FUNCTION_BLOCK ConveyorCTLRing (* Basic Function Block Type *)
  (* Standard: 61499-2 *)
  (* Version 0.2, 2003-12-04, JHC, Rockwell Automation, Renamed for better indexing. *)
  (* Version 0.1, 2002-11-05, JHC, Rockwell Automation, Corrected missing ST element in Algorithm REQ. *)
  (* Version 0.0, 2000-05-30, JHC, Rockwell Automation *)
  (* Compiler header: package fb.rt.cs725; *)
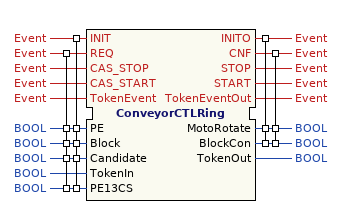
  EVENT_INPUT
    INIT WITH PE, Block, Candidate, PE13CS; (* Initialization Request *)
    REQ WITH PE, Block, Candidate, PE13CS; (* Normal Execution Request *)
    CAS_STOP;
    CAS_START;
    TokenEvent;
  END_EVENT
  EVENT_OUTPUT
    INITO WITH MotoRotate, BlockCon; (* Initialization Confirm *)
    CNF WITH MotoRotate, BlockCon; (* Execution Confirmation *)
    STOP;
    START;
    TokenEventOut;
  END_EVENT
  VAR_INPUT
    PE : BOOL; (* Input event qualifier *)
    Block : BOOL;
    Candidate : BOOL;
    TokenIn : BOOL;
    PE13CS : BOOL;
  END_VAR
  VAR_OUTPUT
    MotoRotate : BOOL; (* Output event qualifier *)
    BlockCon : BOOL;
    TokenOut : BOOL;
  END_VAR
  VAR
    lastPE : BOOL := 1;
    lastBlock : BOOL := 0;
  END_VAR
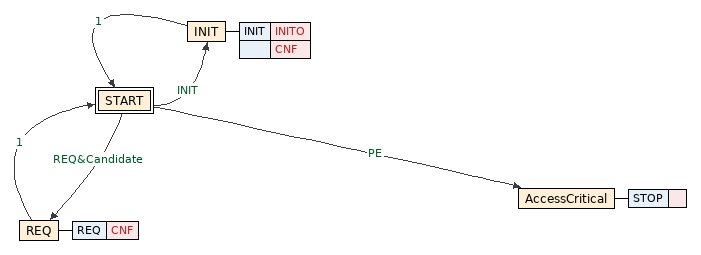
  EC_STATES
    START; (* Initial State *)
    INIT : INIT -> INITO, -> CNF; (* Initialization *)
    REQ : REQ -> CNF; (* Normal execution *)
    AccessCritical : STOP;
  END_STATES
  EC_TRANSITIONS
    START TO INIT := INIT;
    INIT TO START := 1;
    START TO REQ := REQ&Candidate;
    REQ TO START := 1;
    START TO AccessCritical := PE;
  END_TRANSITIONS
  ALGORITHM INIT IN ST: (* Initialization algorithm *)
MotoRotate := TRUE;
Block := FALSE;

System.out.println(this + " " + MotoRotate);
System.out.println(MotoRotate);
  END_ALGORITHM
  ALGORITHM REQ IN Java: (* Normally executed algorithm *)
System.out.println(this+" -> Candidate"+Candidate.value);
if(Candidate.value){
if(lastPE.value!=PE.value){
if(!PE.value){
BlockCon.value=true;
System.out.println("BlockCon = true");
}
else{
BlockCon.value=false;
System.out.println("BlockCon = false");
}
lastPE.value=PE.value;
}
if(lastBlock.value!=Block.value){
if(Block.value){
STOP.serviceEvent(this);
MotoRotate.value=false;
System.out.println("Cas Stop");
}
else{
START.serviceEvent(this);
MotoRotate.value=true;
System.out.println("Cas Start");
}
lastBlock.value=Block.value;
}
}
  END_ALGORITHM
  ALGORITHM START IN Java:
MotoRotate.value=true;
System.out.println(this+" Start "+MotoRotate.value);

System.out.println("Start "+MotoRotate.value);
  END_ALGORITHM
  ALGORITHM STOP IN Java:
MotoRotate.value=false;
System.out.println(this+" Stop "+MotoRotate.value);

System.out.println("Stop "+MotoRotate.value);
  END_ALGORITHM
  ALGORITHM TokenInUse IN Java:
Token.value = false;
  END_ALGORITHM
  ALGORITHM TokenFree IN Java:
Token.value = true;
  END_ALGORITHM
END_FUNCTION_BLOCK
